PROGRAM POU_1
VAR
END_VAR

END_PROGRAM

(* stored: Version 1.1.0.1, ProductVersion 3.1.4024.13
   POU POU_1: Id {125bf085-345b-4d97-b9ac-6266b5141218}, SpecialFunc None *)
